/// Implicitly generated code : DO NOT EDIT!!!
/// Checks for division by 0, if divisor is 0, replace it with 1 and report error
{attribute 'no_check' := ''}
{attribute 'check_div_int64' := ''}
FUNCTION CheckDivLInt : LINT
VAR_INPUT
	divisor: LINT;
END_VAR

IF divisor = 0 THEN
	// replace divisor and report error if necessary
	CheckDivLInt := 1;
	Services.fbEventHandler.Select(TC_Events.CodeEventClass.ErrorEvent)
						   .ArgSetString('div 0 LINT')
						   .Raise();
ELSE
	CheckDivLInt := divisor;
END_IF;

END_FUNCTION

(* stored: Version 1.1.0.1
   POU CheckDivLInt: Id {d92deee1-0768-4838-8012-fc174f42ccd6}, SpecialFunc None *)
